//{attribute 'TcCallAfterOutputUpdate' }
PROGRAM gapUpdate
VAR
    fbCalcGap1 : FB_CalculateGap;
    //FB Variables for Muon Gates
    StateMachine: INT;
    i : UINT;
    fPositionToSet : LREAL;
    toggleExecute : BOOL;
    fCalculatedPosition AT %Q*: REAL;
    fCalculatedInt AT %Q* : DINT;
END_VAR

fbCalcGap1.AngleBladeA := GVL.astAxes[1].stStatus.fActPosition;
fbCalcGap1.AngleBladeB := GVL.astAxes[2].stStatus.fActPosition;
fbCalcGap1();
fCalculatedPosition:= fbCalcGap1.GapSize;
fCalculatedPosition:= fCalculatedPosition*10000;
fCalculatedInt:=  REAL_TO_DINT(fCalculatedPosition);

END_PROGRAM

(* stored: Version 1.1.0.1, ProductVersion 3.1.4024.3
   POU gapUpdate: Id {052ae45b-4e00-406b-8780-3da133e30d51}, SpecialFunc None *)
